TYPE ST_HardwareProcData :
STRUCT
	nHardwareId		: DINT;		//4Byte
	nValue			: DINT;		//4Byte
	nInterpretation	: DINT;		//4Byte
END_STRUCT
END_TYPE

(* stored: Version 1.1.0.1, ProductVersion 3.1.0.25
   DUT ST_HardwareProcData: Id {85d9bb2d-76aa-4dd1-b8a3-68a789847ead} *)
